(* IEC 61131-3 sources: StewartPlatform/Class/SCP111, 1 file *)

(* ---- SCP111.st ---- *)
#define SCP111_DEVICE_ID 1049

(*!
<Class
	Name               = "SCP111"
	Revision           = "1.10"
	RealtimeTask       = "false"
	CyclicTask         = "false"
	BackgroundTask     = "false"
	Sigmatek           = "true"
	OSInterface        = "false"
	HighPriority       = "false"
	Automatic          = "false"
	UpdateMode         = "Prescan"
	IconPath           = ".\Class\scp.ico"
	SharedCommandTable = "true"
	Objectsize         = "(670,120)"
	Comment            = "Class for an SCP111 Safety-Modul">
	<Channels>
		<Server Name="CanOut" Visualized="false" Initialize="false" WriteProtected="true" Retentive="false"/>
		<Server Name="ClassState">
		</Server>
		<Server Name="DesignerPrjConfigCRC" Visualized="false" Initialize="false" WriteProtected="true" Retentive="false" Comment="Shows the CRC of the SafetyDesigner project.&#13;&#10;Compare this with the CRC shown in the SafetyDesigner when printing the project (in the preview or on paper)"/>
		<Server Name="DesignerPrjName" Class="String" Visualized="true" Initialize="false" WriteProtected="true" Retentive="false" Comment="shows the name of the actual safety designer project"/>
		<Server Name="DesignerPrjRev" Class="String" Visualized="true" Initialize="false" WriteProtected="true" Retentive="false" Comment="shows the revision of the actual safety designer project"/>
		<Server Name="ErrorState" Visualized="true" Initialize="false" WriteProtected="true" Retentive="false" Comment="0: no error&#13;&#10;1: error&#13;&#10;2: communication timeout on input data from other safety modules"/>
		<Server Name="FastUnsafeInputs" Visualized="true" Initialize="true" WriteProtected="false" Retentive="false" Comment="write the 32 fast unsafe inputs to this server (bit coded)"/>
		<Server Name="FastUnsafeOutputs" Visualized="true" Initialize="false" WriteProtected="false" Retentive="false" Comment="this server shows the actual state of the 32 fast unsafe outputs (bit coded)"/>
		<Server Name="FirmwareVersion" Visualized="true" Initialize="false" WriteProtected="true" Retentive="false" Comment="Firmware version&#13;&#10;&#13;&#10;Format:&#13;&#10;16#XXXXYYYY&#13;&#10;&#13;&#10;XXXX = Major Revision&#13;&#10;YYYY = Minor Revision"/>
		<Server Name="GetDiagConnect" Visualized="false" Initialize="false" WriteProtected="true" Retentive="false"/>
		<Server Name="QuitComError" Visualized="true" Initialize="false" WriteProtected="false" Retentive="false" Comment="Write to this server to quit communication errors (indicated if Server ErrorState = 2)&#13;&#10;This server can also quit general errors (Server ErrorState = 1) if the safety.dlm is used.&#13;&#10;&#13;&#10;To detect the used quit method, read the server directly after writing. In both cases the error quitting is done asynchronously (= not immediately).&#13;&#10;&#13;&#10;Server shows actual quit-state&#13;&#10;  2..busy with quitting general errors (safety dll version 6 or higher required)&#13;&#10;  1..busy with quitting communication error&#13;&#10;  0..ready&#13;&#10; -1..error at creating a new safety state&#13;&#10; -2..failed to disable user prompt for quit error&#13;&#10; -3..failed to select module via safety number&#13;&#10; -4..error at establishing connection to module (safety designer must not be online at the same time!)&#13;&#10; -5..failed to send the quit error command to the module&#13;&#10; -6..failed to delete the created safety state"/>
		<Server Name="RunState" Visualized="true" Initialize="false" WriteProtected="true" Retentive="false" Comment="0: not running&#13;&#10;1: running in operational or temporary operational mode"/>
		<Server Name="SafetyNumber" Visualized="true" Initialize="false" WriteProtected="true" Retentive="false" Comment="Shows the unique safety number of this module"/>
		<Server Name="SafetyRetryCounter" Visualized="true" Initialize="false" WriteProtected="true" Retentive="false" Comment="Shows the amount of all retries on the safety bus."/>
		<Server Name="SafetyState" Visualized="true" Initialize="false" WriteProtected="true" Retentive="false" Comment="Shows state of safety module&#13;&#10;&#13;&#10;_ModuleNotFound:&#13;&#10; - Module has not been found at the given position&#13;&#10;&#13;&#10;_WaitForSynchronicity:&#13;&#10; - Waiting to get synchrony with interacting modules&#13;&#10;&#13;&#10;_SafetyClassOK:&#13;&#10; - Module has been found and no errors reported&#13;&#10;&#13;&#10;_MemAllocFailed: &#13;&#10; - Failed to allocate or reallocate some memory for the module&#13;&#10;&#13;&#10;_ReadFWVerFailed:&#13;&#10; - Failed to read firmware version of module&#13;&#10;&#13;&#10;_ReinitConfig:&#13;&#10; - Only for CPU: Config of CPU has changed and update is in progress&#13;&#10;&#13;&#10;_ModFromCfgNotFound (Only for CPU):&#13;&#10; - Module in configuration, which is not physically available and HW-Class is placed&#13;&#10; - Module in configuration, which is not physically available and no HW-Class is placed&#13;&#10; - Module in configuration, which is not a CDIAS module (according to it&apos;s HW-Path)&#13;&#10;&#13;&#10;_UnsafeVarNotFound (Only for CPU):&#13;&#10; - Couldn&apos;t find an unsafe variable in the project. Compare spelling in Designer and in project.&#13;&#10;&#13;&#10;_UnknownCfgError (Only for CPU):&#13;&#10; - Error in reading config or creating routing tables occured.&#13;&#10;&#13;&#10;_AsyncComError: &#13;&#10; - Too many consecutive asynchronous commands failed! Please contact Sigmatek Support! &#13;&#10; &#13;&#10;_DOsIncreasedRestartApp: &#13;&#10; - Number or size of module accesses increased with new safety project! &#13;&#10; - =&gt; Can&apos;t continue, because the new data is not covered by the actual accesses! Restart Application! &#13;&#10; &#13;&#10;_LostPowerSupply: &#13;&#10; - The power supply of the safe CPU has been lost. &#13;&#10; &#13;&#10;_WrongSafetyHW: &#13;&#10; - The Safety objects in the project do not match the physical modules. &#13;&#10; - For every physical module a safety object must be placed in the project!"/>
		<Server Name="SdiasSafetyOut" Visualized="true" Initialize="false" WriteProtected="true" Retentive="false"/>
		<Server Name="ServiceMode" Visualized="true" Initialize="false" WriteProtected="true" Retentive="false" Comment="0: operational mode&#13;&#10;1: service mode or temporary operational mode&#13;&#10;2: check configuration phase"/>
		<Server Name="ValidationButtonState" Visualized="true" Initialize="false" WriteProtected="true" Retentive="false" Comment="Shows the state of the validation button&#13;&#10;0: Validation button not used at the moment&#13;&#10;1: Select a command by pressing the button&#13;&#10;2: Command is executed&#13;&#10;3: Error in module"/>
		<Client Name="SdiasSafetyManagerFSoE1" Required="true" Internal="true"/>
		<Client Name="ServerUpdateTime" Required="false" Internal="false" Comment="Time in ms, how long the Servers (unsafe variables in Safety Designer) should take to update.&#13;&#10;This Client is automatically updated, if the given time is too short to handle with the current amount of servers."/>
	</Channels>
	<RevDoku>
		<Owner Company="Sigmatek" Author="RamAnd"/>
		<Dokumentation Revision="1.10" Date="12.07.2016" Author="SeiChr" Company="Sigmatek" Description="Added Values for the total Current calculation. SA 31571"/>
		<Dokumentation Revision="1.9" Date="04.07.2016" Author="RamAnd" Company="Sigmatek" Description="It&apos;s now allowed to have an object of an IO module or HBG if it&apos;s not set to required and it&apos;s neither projected in the safety designer nor physically available."/>
		<Dokumentation Revision="1.8" Date="08.03.2016" Author="EisMic" Company="Sigmatek" Description="Added support for SafetyDiagnosisInfo hardwareclass."/>
		<Dokumentation Revision="1.7" Date="21.01.2016" Author="EisMic" Company="Sigmatek" Description="Outputs are now written in RtPostScan instead of RtPreScan to improve the reaction speed.&#13;&#10;LED-stati are now set to the right state if the SCP is used without any I/O modules."/>
		<Dokumentation Revision="1.6" Date="31.08.2015" Author="RamAnd" Company="Sigmatek" Description="If no configuration is available at the CPU, the optional settings are now ignored since they are not available in this state. This could have lead to SDIAS errors if safety modules were set to required."/>
		<Dokumentation Revision="1.5" Date="31.07.2015" Author="RamAnd" Company="Sigmatek" Description="Added server DesignerPrjConfigCRC to show the CRC of the SafetyDesigner project.&#13;&#10;Added support for optional Safe-IOs (configured in SafetyDesigner)."/>
		<Dokumentation Revision="1.4" Date="22.06.2015" Author="EisMic" Company="Sigmatek" Description="The servers FPGAVersion, SerialNo, Device ID and status and input servers are now not reset anymore when the module is disconnected."/>
		<Dokumentation Revision="1.3" Date="08.06.2015" Author="PieSte" Company="Sigmatek" Description="Changes at Lhd-file for &quot;TypeId&quot; were not taken over."/>
		<Dokumentation Revision="1.2" Date="21.05.2015" Author="PieSte" Company="Sigmatek" Description="Corrected spelling attribute &quot;TypeId&quot; at lhd-file."/>
		<Dokumentation Revision="1.1" Date="16.04.2015" Author="EisMic" Company="Sigmatek" Description="Added support for graphical hardware editor."/>
		<Dokumentation Revision="1.0" Date="15.04.2015" Author="RamAnd" Company="Sigmatek" Description="First library version"/>
	</RevDoku>
	<Network Name="SCP111">
		<!-- List of Components in this network -->
		<Components>
			<Object
				Name       = "_base"
				Class      = "BusInterfaceSdias"
				Position   = "(218,120)"
				Visualized = "true">
				<Channels>
					<Server Name="CallCommand"/>
					<Server Name="ClassState"/>
					<Server Name="DeviceID"/>
					<Server Name="FPGAVersion"/>
					<Server Name="HwVersion"/>
					<Server Name="LEDControl" Value="0"/>
					<Server Name="RetryCounter"/>
					<Server Name="SerialNo"/>
					<Client Name="Place" Value="0"/>
					<Client Name="Required" Value="1"/>
					<Client Name="SdiasIn"/>
				</Channels>
			</Object>
			<Object
				Name           = "SdiasSafetyManagerFSoE1"
				Class          = "SdiasSafetyManagerFSoE"
				Position       = "(990,570)"
				Visualized     = "true"
				BackgroundTime = "100 ms">
				<Channels>
					<Server Name="CanOut"/>
					<Server Name="ClassSvr"/>
					<Server Name="DesignerPrjConfigCRC"/>
					<Server Name="DesignerPrjName"/>
					<Server Name="DesignerPrjRev"/>
					<Server Name="ErrorState"/>
					<Server Name="FastUnsafeInputs"/>
					<Server Name="FastUnsafeOutputs"/>
					<Server Name="FirmwareVersion"/>
					<Server Name="GetDiagConnect"/>
					<Server Name="QuitComError"/>
					<Server Name="RunState"/>
					<Server Name="SafetyNumber"/>
					<Server Name="SafetyRetryCounter"/>
					<Server Name="SafetyState"/>
					<Server Name="SdiasSafetyOut"/>
					<Server Name="ServiceMode"/>
					<Server Name="ValidationButtonState"/>
					<Server Name="VoltageOK"/>
					<Client Name="DeviceID" Value="SCP111_DEVICE_ID"/>
					<Client Name="ServerUpdateTime" Value="50"/>
					<Client Name="ToBusInterface"/>
				</Channels>
			</Object>
		</Components>
		<Comments>
		</Comments>
		<!-- List of Connections in this network -->
		<Connections>
			<Connection Source="this.ClassState" Destination="_base.ClassState" Vertices="(1848,210),(736,210),"/>
			<Connection Source="this.DeviceID" Destination="_base.DeviceID" Vertices="(1848,270),(736,270),"/>
			<Connection Source="this.SerialNo" Destination="_base.SerialNo" Vertices="(1848,390),(736,450),"/>
			<Connection Source="this.RetryCounter" Destination="_base.RetryCounter" Vertices="(1848,450),(736,510),"/>
			<Connection Source="this.SdiasSafetyOut" Destination="SdiasSafetyManagerFSoE1.SdiasSafetyOut" Vertices="(1848,1290),(1676,1680),"/>
			<Connection Source="SdiasSafetyManagerFSoE1.ServerUpdateTime" Destination="this.ServerUpdateTime" Vertices="(990,720),(38,510),"/>
			<Connection Source="this.FPGAVersion" Destination="_base.FPGAVersion" Vertices="(1848,330),(736,330),"/>
			<Connection Source="this.SafetyState" Destination="SdiasSafetyManagerFSoE1.SafetyState" Vertices="(1848,510),(1676,720),"/>
			<Connection Source="_base.SdiasIn" Destination="this.SdiasIn" Vertices="(218,210),(38,210),"/>
			<Connection Source="_base.Place" Destination="this.Place" Vertices="(218,270),(38,270),"/>
			<Connection Source="_base.Required" Destination="this.Required" Vertices="(218,330),(38,330),"/>
			<Connection Source="this.QuitComError" Destination="SdiasSafetyManagerFSoE1.QuitComError" Vertices="(1848,750),(1676,1020),"/>
			<Connection Source="this.FirmwareVersion" Destination="SdiasSafetyManagerFSoE1.FirmwareVersion" Vertices="(1848,810),(1676,1080),"/>
			<Connection Source="this.SafetyNumber" Destination="SdiasSafetyManagerFSoE1.SafetyNumber" Vertices="(1848,870),(1676,1140),"/>
			<Connection Source="this.DesignerPrjName" Destination="SdiasSafetyManagerFSoE1.DesignerPrjName" Vertices="(1848,990),(1676,1380),"/>
			<Connection Source="this.DesignerPrjRev" Destination="SdiasSafetyManagerFSoE1.DesignerPrjRev" Vertices="(1848,1050),(1676,1440),"/>
			<Connection Source="this.CanOut" Destination="SdiasSafetyManagerFSoE1.CanOut" Vertices="(1848,1350),(1676,1740),"/>
			<Connection Source="this.SafetyRetryCounter" Destination="SdiasSafetyManagerFSoE1.SafetyRetryCounter" Vertices="(1848,1410),(1676,1200),"/>
			<Connection Source="this.SdiasSafetyManagerFSoE1" Destination="SdiasSafetyManagerFSoE1.ClassSvr"/>
			<Connection Source="SdiasSafetyManagerFSoE1.ToBusInterface" Destination="_base.CallCommand" Vertices="(990,660),(736,630),"/>
			<Connection Source="this.DesignerPrjConfigCRC" Destination="SdiasSafetyManagerFSoE1.DesignerPrjConfigCRC" Vertices="(1848,930),(1676,1260),"/>
			<Connection Source="this.GetDiagConnect" Destination="SdiasSafetyManagerFSoE1.GetDiagConnect" Vertices="(1848,1470),(1676,1320),"/>
		</Connections>
		<!-- Headerfiles -->
		<Options>
		</Options>
	</Network>
</Class>
*)
#pragma using BusInterfaceSdias

SCP111 : CLASS
: BusInterfaceSdias
  //Servers:
	SafetyState 	: SvrCh_SafetyConfigStateType;
	RunState 	: SvrCh_DINT;
	ServiceMode 	: SvrCh_DINT;
	ErrorState 	: SvrCh_DINT;
	QuitComError 	: SvrCh_DINT;
	FirmwareVersion 	: SvrCh_HDINT;
	SafetyNumber 	: SvrCh_HDINT;
	DesignerPrjConfigCRC 	: SvrCh_HDINT;
	DesignerPrjName 	: SvrChCmd_UDINT;
	DesignerPrjRev 	: SvrChCmd_UDINT;
	ValidationButtonState 	: SvrCh_DINT;
	FastUnsafeInputs 	: SvrCh_BDINT;
	FastUnsafeOutputs 	: SvrCh_BDINT;
	SdiasSafetyOut 	: SvrChCmd_DINT;
	CanOut 	: SvrChCmd_DINT;
	SafetyRetryCounter 	: SvrCh_DINT;
	GetDiagConnect 	: SvrChCmd_DINT;
  //Clients:
	ServerUpdateTime 	: CltCh_UDINT;
	SdiasSafetyManagerFSoE1 	: CltChCmd_SdiasSafetyManagerFSoE;
  //Variables:
  //Functions:

	FUNCTION VIRTUAL GetDeviceID
		VAR_OUTPUT
			output 	: UDINT;
		END_VAR;
				//! <Function Comment="Make a request to fetch the diagnosis data" Name="FetchDiagState"/>
	FUNCTION VIRTUAL GLOBAL FetchDiagState;
				//! <Function Comment="Check if the diagnosis data have arrived (if so, retcode = TRUE)." Name="GetDiagState"/>
	FUNCTION VIRTUAL GLOBAL GetDiagState
		VAR_INPUT
			pDiagState 	: ^SafetyDiagState;
		END_VAR
		VAR_OUTPUT
			StateReady 	: BOOL;			//! <Variable Comment="FALSE...State is not ready (value of &quot;input parameter&quot; not changed)&#13;&#10;TRUE....State is ready (input parameter)" Name="GetDiagState.StateReady"/>
		END_VAR;

	FUNCTION VIRTUAL GLOBAL FetchDiagInfo
		VAR_INPUT
			ucChoice 	: USINT;			//! <Variable Comment="   0..µC1&#13;&#10;&lt;&gt; 0..µC2" Name="FetchDiagInfo.ucChoice"/>
		END_VAR;

	FUNCTION VIRTUAL GLOBAL GetDiagInfo
		VAR_INPUT
			pDiagInfo 	: ^SafetyDiagInfo;
		END_VAR
		VAR_OUTPUT
			StateReady 	: BOOL;
		END_VAR;

	FUNCTION VIRTUAL GLOBAL ClassState::NewInst
		VAR_INPUT
			pPara 	: ^CmdStruct;
			pResult 	: ^results;
		END_VAR
		VAR_OUTPUT
			ret_code 	: iprStates;
		END_VAR;

	FUNCTION VIRTUAL GLOBAL SafetyState::Read
		VAR_OUTPUT
			output (EAX) 	: SafetyConfigStateType;
		END_VAR;

	FUNCTION VIRTUAL GLOBAL QuitComError::Read
		VAR_OUTPUT
			output (EAX) 	: DINT;
		END_VAR;

	FUNCTION VIRTUAL GLOBAL QuitComError::Write
		VAR_INPUT
			input (EAX) 	: DINT;
		END_VAR
		VAR_OUTPUT
			result (EAX) 	: DINT;
		END_VAR;

	FUNCTION VIRTUAL GLOBAL FirmwareVersion::Read
		VAR_OUTPUT
			output (EAX) 	: HDINT;
		END_VAR;

	FUNCTION VIRTUAL GLOBAL SafetyNumber::Read
		VAR_OUTPUT
			output (EAX) 	: HDINT;
		END_VAR;

	FUNCTION VIRTUAL GLOBAL DesignerPrjConfigCRC::Read
		VAR_OUTPUT
			output (EAX) 	: HDINT;
		END_VAR;

	FUNCTION VIRTUAL GLOBAL FastUnsafeInputs::Write
		VAR_INPUT
			input (EAX) 	: BDINT;
		END_VAR
		VAR_OUTPUT
			result (EAX) 	: BDINT;
		END_VAR;

	FUNCTION VIRTUAL GLOBAL FastUnsafeOutputs::Write
		VAR_INPUT
			input (EAX) 	: BDINT;
		END_VAR
		VAR_OUTPUT
			result (EAX) 	: BDINT;
		END_VAR;

	FUNCTION VIRTUAL GLOBAL SafetyRetryCounter::Read
		VAR_OUTPUT
			output (EAX) 	: DINT;
		END_VAR;

	FUNCTION VIRTUAL GLOBAL GetDiagConnect::Read
		VAR_OUTPUT
			output (EAX) 	: DINT;
		END_VAR;
  //Tables:
	FUNCTION @STD
		VAR_OUTPUT
			ret_code	: CONFSTATES;
		END_VAR;
	FUNCTION GLOBAL TAB @CT_;
END_CLASS;

#pragma using SdiasSafetyManagerFSoE

FUNCTION VIRTUAL GLOBAL SCP111::SafetyState::Read
	VAR_OUTPUT
		output (EAX) 	: SafetyConfigStateType;
	END_VAR

	SafetyState := SdiasSafetyManagerFSoE1.SafetyState.Read();
	output := SafetyState;

END_FUNCTION

FUNCTION VIRTUAL GLOBAL SCP111::QuitComError::Read
	VAR_OUTPUT
		output (EAX) 	: DINT;
	END_VAR

	QuitComError := SdiasSafetyManagerFSoE1.QuitComError.Read();
	output := QuitComError;

END_FUNCTION

FUNCTION VIRTUAL GLOBAL SCP111::QuitComError::Write
	VAR_INPUT
		input (EAX) 	: DINT;
	END_VAR
	VAR_OUTPUT
		result (EAX) 	: DINT;
	END_VAR

	QuitComError := input;
	result := SdiasSafetyManagerFSoE1.QuitComError.Write(QuitComError);

END_FUNCTION

FUNCTION VIRTUAL GLOBAL SCP111::FirmwareVersion::Read
	VAR_OUTPUT
		output (EAX) 	: HDINT;
	END_VAR

	FirmwareVersion := SdiasSafetyManagerFSoE1.FirmwareVersion.Read();
	output := FirmwareVersion;

END_FUNCTION

FUNCTION VIRTUAL GLOBAL SCP111::SafetyNumber::Read
	VAR_OUTPUT
		output (EAX) 	: HDINT;
	END_VAR

	SafetyNumber := SdiasSafetyManagerFSoE1.SafetyNumber.Read();
	output := SafetyNumber;

END_FUNCTION

FUNCTION VIRTUAL GLOBAL SCP111::FastUnsafeInputs::Write
	VAR_INPUT
		input (EAX) 	: BDINT;
	END_VAR
	VAR_OUTPUT
		result (EAX) 	: BDINT;
	END_VAR

	FastUnsafeInputs := input;
	result := SdiasSafetyManagerFSoE1.FastUnsafeInputs.Write(FastUnsafeInputs);

END_FUNCTION

FUNCTION VIRTUAL GLOBAL SCP111::ClassState::NewInst
	VAR_INPUT
		pPara 	: ^CmdStruct;
		pResult 	: ^results;
	END_VAR
	VAR_OUTPUT
		ret_code 	: iprStates;
	END_VAR
  VAR
  	pRtRefreshData : ^t_RtRefresh;
  END_VAR

	ret_code := READY;

	CASE pPara^.uiCmd OF
//**********************************************************************************************************************************************************
		SDIAS_SET_RT_DATA:
      pRtRefreshData        := pPara^.aPara[0]$^t_RtRefresh;
      RunState              := pRtRefreshData^.LEDRunState;
      ServiceMode           := pRtRefreshData^.LEDServiceMode;
      ErrorState            := pRtRefreshData^.LEDErrorState;
      ValidationButtonState := pRtRefreshData^.LEDValidationButtonState;
      FastUnsafeOutputs     := pRtRefreshData^.FastUnsafeOutputs;

//**********************************************************************************************************************************************************
		SDIAS_SET_SAFETY_STATE:
      SafetyState := pPara^.aPara[0]$SafetyConfigStateType;

//**********************************************************************************************************************************************************
		SDIAS_SET_ASY_STATE:
      QuitComError := pPara^.aPara[0]$^t_AsyRefresh^.QuitComError;

//**********************************************************************************************************************************************************

  ELSE
    ret_code := BusInterfaceSdias::ClassState::NewInst(pPara, pResult);
	END_CASE;

END_FUNCTION

FUNCTION VIRTUAL GLOBAL SCP111::FastUnsafeOutputs::Write
	VAR_INPUT
		input (EAX) 	: BDINT;
	END_VAR
	VAR_OUTPUT
		result (EAX) 	: BDINT;
	END_VAR

	result := SdiasSafetyManagerFSoE1.FastUnsafeOutputs.Write(input);

END_FUNCTION

FUNCTION VIRTUAL GLOBAL SCP111::SafetyRetryCounter::Read
	VAR_OUTPUT
		output (EAX) 	: DINT;
	END_VAR

	SafetyRetryCounter := SdiasSafetyManagerFSoE1.SafetyRetryCounter.Read();
	output := SafetyRetryCounter;

END_FUNCTION

FUNCTION VIRTUAL SCP111::GetDeviceID
	VAR_OUTPUT
		output 	: UDINT;
	END_VAR

  output := SCP111_DEVICE_ID;

END_FUNCTION

FUNCTION VIRTUAL GLOBAL SCP111::FetchDiagState

  SdiasSafetyManagerFSoE1.FetchDiagState();

END_FUNCTION

FUNCTION VIRTUAL GLOBAL SCP111::GetDiagState
	VAR_INPUT
		pDiagState 	: ^SafetyDiagState;
	END_VAR
	VAR_OUTPUT
		StateReady 	: BOOL;
	END_VAR

  StateReady := SdiasSafetyManagerFSoE1.GetDiagState(pDiagState);

END_FUNCTION

FUNCTION VIRTUAL GLOBAL SCP111::FetchDiagInfo
	VAR_INPUT
		ucChoice 	: USINT;
	END_VAR

  SdiasSafetyManagerFSoE1.FetchDiagInfo(ucChoice);

END_FUNCTION

FUNCTION VIRTUAL GLOBAL SCP111::GetDiagInfo
	VAR_INPUT
		pDiagInfo 	: ^SafetyDiagInfo;
	END_VAR
	VAR_OUTPUT
		StateReady 	: BOOL;
	END_VAR

  StateReady := SdiasSafetyManagerFSoE1.GetDiagInfo(pDiagInfo);

END_FUNCTION

FUNCTION VIRTUAL GLOBAL SCP111::DesignerPrjConfigCRC::Read
	VAR_OUTPUT
		output (EAX) 	: HDINT;
	END_VAR

	DesignerPrjConfigCRC := SdiasSafetyManagerFSoE1.DesignerPrjConfigCRC.Read();
	output := DesignerPrjConfigCRC;

END_FUNCTION

FUNCTION VIRTUAL GLOBAL SCP111::GetDiagConnect::Read
	VAR_OUTPUT
		output (EAX) 	: DINT;
	END_VAR

	GetDiagConnect := SdiasSafetyManagerFSoE1.GetDiagConnect.Read();
	output := GetDiagConnect;

END_FUNCTION
